TYPE DUT_SENSOR_DATAS_7 :
UNION
	data_lreal:REAL;
	data_byte:ARRAY[0..3] OF BYTE;
END_UNION
END_TYPE

(* stored: Version 1.1.0.1, ProductVersion 3.1.4024.6
   DUT DUT_SENSOR_DATAS_7: Id {9855b516-318f-4cb9-9dde-d38f77fd9cef} *)
